Universal Robots PolyScope program: vert path wp save.urp

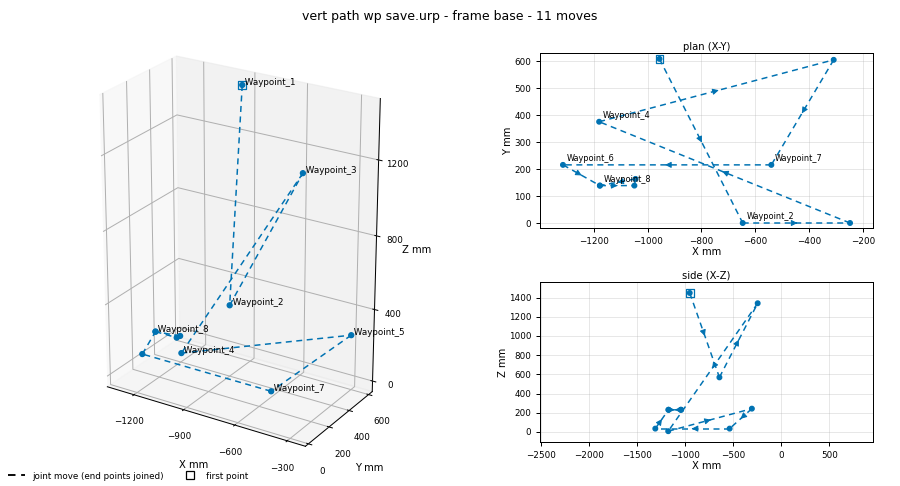
[picture p0: tool path of vert path wp save.urp in frame base, 11 of 11 moves have a stored position in this frame; points joined in program order, loops and branches not executed]
Program vert path wp save (installation=munsch directory=/programs createdIn=5.14.5 lastSavedIn=5.14.5 robotSerialNumber=20236801216)
Calibrated DH parameters: a=[-0.000021, -0.748897, -0.28186, -0.00004, -0.000055, 0]; d=[0.236225, -424.082933, -1564.66872, 1988.95162, 0.159094, 0.153873]; alpha=[1.570844, 0.001002, 0.000337, 1.571488, -1.569996, 0]; deltaTheta=[0, -0.516316, 5.626292, 1.173211, 0.000001, 0]
InitVariablesNode
Robot Program (runOnlyOnce=false)
  SafeHome (positionOptionType=SPEED_AND_ACCELERATION speed=1.047198 acceleration=1.396263 nextMotionTime=2)
  MoveJ speed 60 deg/s, acceleration 80 deg/s^2 (useActiveTCP=true) feature=Base
    Waypoint Waypoint_1: motionParameters(nextMotionTime=2); TCP in base x=-955.652 y=609.645 z=1447.607 mm, rx=0 ry=0 rz=0 rad; joints [-35.47, -19.301, -23.677, 222.924, 125.529, -0.027] deg; TCP offset x=8.55 y=-271.52 z=102 mm, rx=1.2092 ry=-1.2092 rz=1.2092 rad
    Waypoint Waypoint_2: TCP in base x=-646.472 y=-0.005 z=568.192 mm, rx=0 ry=0 rz=0 rad; joints [-13.368, 55.623, -112.874, 237.203, 103.359, -0.015] deg
    Waypoint Waypoint_3: TCP in base x=-247.842 y=-0.001 z=1340.099 mm, rx=1.5708 ry=0 rz=0 rad; joints [-48.812, -19.022, -93.44, 292.414, 138.853, 89.976] deg
  MoveJ speed 60 deg/s, acceleration 80 deg/s^2 (useActiveTCP=true) feature=Base
    Waypoint Waypoint_4: TCP in base x=-1179.747 y=376.142 z=7.543 mm, rx=1.38 ry=-0.892 rz=-0.892 rad; joints [-43.861, -14.749, 70.025, 124.69, 68.156, 89.98] deg
    Waypoint Waypoint_5: TCP in base x=-308.519 y=606.107 z=242.384 mm, rx=-2.1337 ry=0.3495 rz=2.1309 rad; joints [-106.377, -74.131, 126.549, 42.484, 90.905, 87.285] deg
    Waypoint Waypoint_7: TCP in base x=-540.146 y=215.928 z=34.627 mm, rx=-1.5058 ry=1.0576 rz=1.5735 rad; joints [-25.658, -64.434, 142.415, 9.313, 85.709, 219.638] deg
    Waypoint Waypoint_6: TCP in base x=-1314.145 y=215.925 z=34.627 mm, rx=-1.5058 ry=1.0576 rz=1.5735 rad; joints [-8.569, -32.934, 66.275, 52.815, 86.649, 236.732] deg
  MoveJ speed 60 deg/s, acceleration 80 deg/s^2 (useActiveTCP=true) feature=Base
    Waypoint Waypoint_8: TCP in base x=-1176.984 y=138.952 z=230.662 mm, rx=-0.853 ry=-1.646 rz=1.646 rad; joints [-20.645, -63.464, 120.754, 302.711, 124.07, 90.04] deg; TCP offset x=-4.211 y=-279.829 z=105.916 mm, rx=1.2092 ry=-1.2092 rz=1.2092 rad
    Waypoint Waypoint_9: TCP in base x=-1048.769 y=138.957 z=230.694 mm, rx=-0.853 ry=-1.646 rz=1.646 rad; joints [-24.627, -68.929, 131.421, 297.5, 120.091, 90.036] deg
    Waypoint Waypoint_10: TCP in base x=-1044.593 y=163.806 z=230.713 mm, rx=-0.8978 ry=-1.6009 rz=1.6009 rad; joints [-24.627, -68.929, 131.421, 297.5, -236.127, 90.036] deg
    Waypoint Waypoint_11: TCP in base x=-1177 y=138.945 z=230.679 mm, rx=-0.852 ry=-1.646 rz=1.646 rad; joints [-20.652, -63.452, 120.769, 302.639, -235.955, 90.036] deg
